// TIA Portal V20 export
TYPE "typeIntConditionHmiInterface"
// stored: Access Published, Namespace Unit1.Em2
   STRUCT
      Axis_01 { S7_SetPoint := 'True'} : "LER_typeAxisIntlockAll";   // AnodeMainPnP1AxisX
      Axis_02 { S7_SetPoint := 'True'} : "LER_typeAxisIntlockAll";   // AnodeMainPnP2AxisX
      Axis_03 { S7_SetPoint := 'True'} : "LER_typeAxisIntlockAll";   // AnodeMainPnP1AxisY
      Axis_04 { S7_SetPoint := 'True'} : "LER_typeAxisIntlockAll";   // AnodeMainPnP1AxisZ
      Actuator_15 { S7_SetPoint := 'True'} : "LER_typeAxisActuatorCondition";   // AnodeNgBoxLockUpDown
      Actuator_16 { S7_SetPoint := 'True'} : "LER_typeAxisActuatorCondition";   // AnodeMaintenanceMovingFixFrontFwdBwd
   END_STRUCT;
END_TYPE
